(* IEC 61131-3 sources: plc-home-automation/home_automation/lighting_heating_updated, 19 files *)

(* ---- AlarmGlobals.st ---- *)
VAR_GLOBAL CONSTANT

   C_FRONT_DOOR_OPENING : INT := 1;
   C_GARAGE_DOOR_OPENING : UINT   := 2;
   C_HALL_ZONE : UINT        := 4;
   C_GARAGE_ZONE : UINT          := 5;
   C_KITCHEN_ZONE : UINT          := 6;
   C_LIVING_ROOM_ZONE : UINT         := 7;
   C_BEDROOM_ZONE : UINT            := 8;
   C_DOWNSTAIRS_BATH_ZONE : UINT      := 9;
   C_HALLWAY_ZONE : UINT         := 10;
   C_CHILDRENS_ROOM_3_ZONE : UINT   := 11;
   C_CHILDRENS_ROOM_1_ZONE : UINT   := 12;
   C_CHILDRENS_ROOM_2_ZONE : UINT   := 13;
   C_UPSTAIRS_BATH_ZONE : UINT     := 14;
   C_WC_ZONE : UINT              := 15;
   C_BOILER_ZONE : UINT           := 16;

   C_UNCONNECTED_NO_OP : UINT    := 3;

   C_ALARM_ZONES : UINT      := 16;
END_VAR

VAR_GLOBAL
    PARADOX_COM : fbPAR_DIG_EVOsystem;
    PARADOX_DATA : T_PAR_DIG_EVO_SYSTEM_DATA;
    ALARM_ZONES_INACTIVITY : ARRAY [1 .. C_ALARM_ZONES] OF BOOL;
    ALARM_ZONES_SABOTAGE : ARRAY [1 .. C_ALARM_ZONES] OF BOOL;
    ALARM_ZONES_ERROR : ARRAY [1 .. C_ALARM_ZONES] OF BOOL;
    ALARM_ACTIVE : BOOL;

    AWAY_TIMER: TON;

    TIME_AWAY_SHORT : TIME := T#20m;
    TIME_AWAY_LONG : TIME := T#60m;
    GONE_FOR_5_MINUTES : BOOL := FALSE;
    GONE_FOR_SHORT_TIME : BOOL := FALSE;
    GONE_FOR_LONG_TIME : BOOL := FALSE;
END_VAR

FUNCTION awayFromHomeFor : bool
  VAR_INPUT
    awayFor : TIME;  (*Tell me if motion sensors are inactive for that time. Max is 20 days.*)
  END_VAR

  IF(AWAY_TIMER.ET < awayFor) THEN
    awayFromHomeFor := false;
  ELSE
    awayFromHomeFor := true;
  END_IF;

END_FUNCTION

(* ---- HeatingGlobals.st ---- *)
VAR_GLOBAL CONSTANT
   // Heating control locals
   C_BEDROOM_INDEX : INT          := 0;
   C_LIVING_ROOM_1_INDEX : INT     := 1;
   C_LIVING_ROOM_2_INDEX : INT     := 2;
   C_LIVING_ROOM_3_INDEX : INT     := 3;
   C_DOWNSTAIRS_BATH_INDEX : INT    := 4;
   C_HALL_INDEX : INT      := 5;
   C_GARAGE_INDEX : INT        := 6;
   C_CHILDRENS_ROOM_1_INDEX : INT := 7;
   C_CHILDRENS_ROOM_2_INDEX : INT := 8;
   C_CHILDRENS_ROOM_3_INDEX : INT := 9;
   C_HALLWAY_INDEX : INT       := 10;
   C_BOILER_INDEX : INT         := 11;
   C_WC_INDEX : INT            := 12;
   C_UPSTAIRS_BATH_INDEX : INT   := 13;

   C_HEATING_ZONES : INT                  := 14;
   C_DOWNSTAIRS_ZONE_MAX_INDEX_PLUS_ONE : INT := 7;

   C_MAXIMUM_HEATING_TEMPERATURE : REAL := 38.0;
   C_MINIMUM_HEATING_TEMPERATURE : REAL := 28.0;

   C_MAXIMUM_HOT_WATER_TEMPERATURE : REAL := 62.0;
   C_MINIMUM_HOT_WATER_TEMPERATURE : REAL := 35.0;

END_VAR

VAR_GLOBAL
    heatingRequests : ARRAY [0 .. C_HEATING_ZONES - 1] OF BOOL;
END_VAR

VAR_GLOBAL
   HEATING_CONTROL_SAMPLING_TIME : TIME := T#10m;
   IPID_K : REAL := 0.0005;
   IPID_TI : REAL := 0.0001;
   IPID_TD : REAL := 12000;
   OVERSHOOT_HISTERESIS : REAL := 0.2;

   HEATING_ENABLE : BOOL := true;
   HOT_WATER_ENABLE : BOOL := true;
   PRESENCE_BASED_HEATING_CONTROL : BOOL := true;
   PRESENCE_BASED_HOT_WATER_ENABLE : BOOL := true;

   FUTOVIZ_TEMPERATURE : REAL              := 30.0;
   HOT_WATER_TEMPERATURE : REAL  := 42.0;

   LIVING_ROOM_DESIRED_TEMPERATURE : REAL       := 22.0;
   BEDROOM_DESIRED_TEMPERATURE : REAL     := 20.5;
   CHILDRENS_ROOM_1_DESIRED_TEMPERATURE : REAL := 22.0;
   CHILDRENS_ROOM_2_DESIRED_TEMPERATURE : REAL := 21.0;
   CHILDRENS_ROOM_3_DESIRED_TEMPERATURE : REAL := 21.0;
   DOWNSTAIRS_BATH_DESIRED_TEMPERATURE : REAL    := 21.0;
   UPSTAIRS_BATH_DESIRED_TEMPERATURE : REAL   := 21.0;
   GARAGE_DESIRED_TEMPERATURE : REAL        := 5.0;
   BOILER_DESIRED_TEMPERATURE : REAL         := 5.0;
   WC_DESIRED_TEMPERATURE : REAL            := 5.0;
   HALLWAY_DESIRED_TEMPERATURE : REAL       := 5.0;
   HALL_DESIRED_TEMPERATURE : REAL      := 21;

   // For testing purposes only
   WC_TEMPERATURE : REAL              := 30.0;
   HALLWAY_TEMPERATURE : REAL         := 30.0;
   BOILER_ROOM_TEMPERATURE : REAL           := 30.0;

   SUM_HEATING_REQUIREMENT : BOOL := false;
   SUM_HEATING_WATER_TEMPERATURE_REQUIREMENT : REAL := 0;

   MEASURED_TEMPERATURES : ARRAY [0 .. C_HEATING_ZONES - 1] OF PTR_TO REAL;
   DESIRED_TEMPERATURES : ARRAY [0 .. C_HEATING_ZONES - 1] OF PTR_TO REAL;
   VALVE_ACTUATORS : ARRAY [0 .. C_HEATING_ZONES - 1] OF PTR_TO BOOL;

   // You can't take the ADR() of a real const global...
   C_50_FOK : REAL := 50.0;
   C_4_FOK : REAL := 4.0;
END_VAR

(* ---- PersistGlobals.st ---- *)
VAR_GLOBAL CONSTANT
    C_REALS_TO_PERSIST : INT      := 18;
    C_BOOLS_TO_PERSIST : INT      := 4;
    C_PERSIST_DIRECTORY_ROOT : STRING := 'PERSIST';
    C_PERSIST_HEATING_IPID_SUBDIR : STRING := '';
    C_PERSIST_HEATING_SUBDIR : STRING := '/HEATING';
    C_PERSIST_ROOM_TEMPERATURE_SUBDIR : STRING := '/ROOMTMP';
    C_PERSIST_BOILER_CONTROL_SUBDIR : STRING := '/BOILERCT';
END_VAR

VAR_GLOBAL
    REALS_TO_PERSIST : ARRAY [1 .. C_REALS_TO_PERSIST] OF PTR_TO REAL;
    REALS_TO_PERSIST_DIRS : ARRAY [1 .. C_REALS_TO_PERSIST] OF STRING;
    REALS_TO_PERSIST_NAMES : ARRAY [1 .. C_REALS_TO_PERSIST] OF STRING;
    BOOLS_TO_PERSIST : ARRAY [1 .. C_BOOLS_TO_PERSIST] OF PTR_TO BOOL;
    BOOLS_TO_PERSIST_DIRS : ARRAY [1 .. C_BOOLS_TO_PERSIST] OF STRING;
    BOOLS_TO_PERSIST_NAMES : ARRAY [1 .. C_BOOLS_TO_PERSIST] OF STRING;
END_VAR

(* ---- VaillantGlobals.st ---- *)
VAR_GLOBAL
  VAILLANT_ACN                   : bool;  (*altered after loading all the data*)
  VAILLANT_HEATING_TEMP          : real;  (*current boiler temperature*)
  VAILLANT_DWH_TEMP              : real;  (*current DHW temperature*)
  VAILLANT_OUTSIDE_TEMP          : real;  (*current outdoor temperature on boiler sensor*)
  VAILLANT_RETURN_WATER_TEMP     : real;  (*current returning temperature (Some boilers don't measure it)*)
  VAILLANT_MODULATION_LEVEL      : usint; (*value of relative burner modulation (0-100%)*)
  VAILLANT_PRESSURE_LEVEL        : real;  (*value of pressure temperature water (0-5 bar)*)
  VAILLANT_BURNERS_RUNNING       : uint;  (*number of burner starts*)
  VAILLANT_HEATING_ACTIVE        : bool;  (*heating is active (heats right now)*)
  VAILLANT_DWH_ACTIVE            : bool;  (*DHW active (heats right now)*)
  VAILANT_DWH_PRESENT            : bool;  (*boiler reports DHW is present*)
  VAILANT_MODULATION_SUPPORT     : bool;  (*boiler supports power modulation*)
  VAILANT_BURNER_ON              : bool;  (*flame on*)
  VAILANT_ERROR                  : bool;  (*boiler has an error*)
  VAILLANT_DIAG_CODE             : uint;  (*diagnostic code boiler (lower byte = error code = upper byte error flags)*)
  VAILANT_COMMUNICATIONO_ERROR   : bool;  (*communication error*)

END_VAR

(* ---- BathroomFanOnOff.st ---- *)
FUNCTION logBathroomFan : INT
VAR_INPUT
    name : STRING;
    rampOn : BOOL;
    feedOn: BOOL;
    out : BOOL;
END_VAR
     SWITCH_TRACKER(name := name
         + ': ramp(' + BOOL_TO_STRING(rampOn)
         + ') feedOn(' + BOOL_TO_STRING(feedOn)
         + ') out(' + BOOL_TO_STRING(out)
         + ')');

    logBathroomFan := 0;
END_FUNCTION

FUNCTION_BLOCK BathroomFanOnOff

  VAR_INPUT CONSTANT
     name : STRING;
  END_VAR

  VAR_INPUT
     timeOn   : TIME;
     feedOn   : BOOL R_EDGE;
     feedOff  : BOOL R_EDGE;
     change   : BOOL R_EDGE;
  END_VAR

  VAR_OUTPUT
     out : BOOL;
  END_VAR

  VAR
     ramp    : TON;
     rampOn  : BOOL := false;
  END_VAR

  IF change THEN
     rampOn := NOT out;
     out := NOT out;
     logBathroomFan(name:= name, feedOn := feedOn, rampOn := rampOn, out := out);
  END_IF;

  IF feedOn THEN
     rampOn := false;
     out := true;
  END_IF;

  IF feedOff AND out THEN
     rampOn := true;
  END_IF;

  ramp(IN := rampOn, PT := timeOn);

  IF ramp.Q THEN
     out := false;
     rampOn := false;
  END_IF;

END_FUNCTION_BLOCK

(* ---- lighting.ST ---- *)
// Helper function block
TYPE
  ControllerArray : ARRAY [0 .. C_LIGHTS_ZONES_COUNT - 1] OF ChangeOnOff;
END_TYPE

FUNCTION_BLOCK TurnOffLightsHelper
  VAR_INPUT
    offSignal : BOOL R_EDGE;
  END_VAR

  VAR_IN_OUT
    controllers : ControllerArray;
  END_VAR

  VAR
    i : INT := 0;
  END_VAR

  IF (offSignal) THEN
    FOR i := 0 TO C_LIGHTS_ZONES_COUNT - 1 DO
      controllers[i](requestOff := offSignal);
    END_FOR;
  END_IF;

END_FUNCTION_BLOCK // Helper function block

PROGRAM LightingControl

  VAR
    domesticHotWaterCirculation_in : OnThenOffPulse;
    garageGate_in : OnThenOffPulse;

    exhaustRequest: BOOL := false;
    wcExhaustDelay : TON;
    wcExhaustDelayTime : TIME := T#4m;
    upstairsBathroomExhaustDelay : TON;
    upstairsBathroomExhaustDelayTime : TIME := T#8m;
    upstairsShowerExhaustDelay : TON;
    upstairsShowerExhaustDelayTime : TIME := T#3m;
    exhaustFan_in : BathroomFanOnOff;
    exhaustFanRuntime : TIME := T#10m;

    lightsKapcsolok : ControllerArray;
    lightsControlBasedOnOccupancy : TurnOffLightsHelper;

    i : INT := 0;

  END_VAR

    KITCHEN_FURNITURE_LIGHTS_OUT := TRUE; // We have the door bell in that socket for now.

    domesticHotWaterCirculation_in(timeOn := T#2m, timeOff := T#20m, onSignal := (KERINTGETES_SWITCH_IN OR KITCHEN_FURNITURE_LIGHTS_IN OR VIRTUAL_CIRCULATION_SWITCH_IN));
    BOILER_PUMP_PLUG_RIGHT := domesticHotWaterCirculation_in.active;
    VIRTUAL_CIRCULATION_SWITCH_IN := FALSE;

    wcExhaustDelay(IN := UPSTAIRS_WC_LIGHTS_OUT, PT := wcExhaustDelayTime);
    upstairsBathroomExhaustDelay(IN := UPSTAIRS_BATH_MAJOR_LIGHTS_OUT, PT := upstairsBathroomExhaustDelayTime);
    upstairsShowerExhaustDelay(IN := UPSTAIRS_BATH_SHOWER_LIGHTS_OUT, PT := upstairsShowerExhaustDelayTime);
    //exhaustRequest := wcExhaustDelay.Q OR upstairsBathroomExhaustDelay.Q OR upstairsShowerExhaustDelay.Q;
    exhaustRequest := FALSE;
    exhaustFan_in(timeOn := exhaustFanRuntime, feedOn := exhaustRequest, feedOff := NOT exhaustRequest, change := EXHAUST_FAN_IN OR VIRTUAL_EXHAUST_FAN_IN, name := 'Elszivo ventillator');
    EXHAUST_FAN_OUT := exhaustFan_in.out;
    VIRTUAL_EXHAUST_FAN_IN := FALSE;

    garageGate_in(onSignal := GARAGE_GATE_IN OR VIRTUAL_GARAGE_DOOR_OPENER, timeOn := T#0.2s, timeOff := T#0.2s);
    GARAGE_GATE_OUT := garageGate_in.active;
    VIRTUAL_GARAGE_DOOR_OPENER := FALSE;

    HALLWAY_LIGHTS_COMBINED_IN := HALLWAY_LIGHTS_IN OR STAIRS_LIGHTS_IN;

    FOR i := 0 TO C_LIGHTS_ZONES_COUNT - 1 DO
        lightsKapcsolok[i](requestChange := ( LIGHTS_INPUTS[i]^ OR VIRTUAL_LIGHTS_INPUTS[i]^) );
        LIGHTS_OUTPUTS[i]^ := lightsKapcsolok[i].output;
        VIRTUAL_LIGHTS_INPUTS[i]^ := FALSE;
    END_FOR;

    lightsControlBasedOnOccupancy( offSignal := (ALARM_ACTIVE AND GONE_FOR_SHORT_TIME), controllers := lightsKapcsolok );

END_PROGRAM

(* ---- LinearHeatController.st ---- *)
FUNCTION_BLOCK LinearHeatController
  VAR_INPUT
    actualTemperature : REAL := 0;
    setpoint : REAL := 0;
    ramp : REAL := 1;
    offset : REAL := 0;
    histeresis : REAL := 0;
  END_VAR
  VAR_OUTPUT
    heatRequest : BOOL := FALSE;
    heatingTemperature : REAL := 0;
  END_VAR

  heatingTemperature := setpoint + ramp * (setpoint - actualTemperature) + offset;

  IF actualTemperature < (setpoint - histeresis) THEN
     heatRequest := true;
  END_IF;
  IF actualTemperature > (setpoint + histeresis) THEN
     heatRequest := FALSE;
  END_IF;
END_FUNCTION_BLOCK

(* ---- PersistFramework.st ---- *)
FUNCTION createDirectory: BOOL
VAR_INPUT
    dirPath: STRING;
END_VAR

VAR
    errorMessage: STRING;

END_VAR

createDirectory := FileExists(fileName := dirPath);
IF NOT createDirectory THEN
  createDirectory := DirCreate(dirName := dirPath);
  IF NOT createDirectory THEN
    GetLastErrTxt( errCode := GetLastErr(), errMessage := errorMessage);
    FILE_PROBLEM_TRACKER(name := 'Dir create error:');
    FILE_PROBLEM_TRACKER(name := dirPath);
    FILE_PROBLEM_TRACKER(name := errorMessage);
    return;
  END_IF;
END_IF;

createDirectory := true;

END_FUNCTION

FUNCTION_BLOCK Persistor

VAR_IN_OUT
    compilerBugPlaceholder: BOOL;
    dirPath: STRING;
    fileName: STRING;
    data : UDINT;
END_VAR
VAR_INPUT
    dataSize: UDINT;
    toWrite : BOOL;
END_VAR
VAR_OUTPUT
    busy: BOOL := FALSE;
END_VAR

VAR
    fullPath : STRING;

    writer  : WriteToFile;
    reader : ReadFromFile;
    reading : BOOL := false;
    writing : BOOL := false;

    errorMessage : STRING;
    file : BOOL;
END_VAR

// Workaround for a compiler bug which renders the address of the first VAR_IN_OUT to the unusable %X0.0 no matter what.
IF FALSE THEN compilerBugPlaceholder := compilerBugPlaceholder; END_IF;

IF writing THEN
    writer( fileName := fullPath,
            srcVar := data,
            exec := writing,
            seek := 0,
            size := dataSize
            );
    writing := writer.busy;
    IF writer.err THEN
      GetLastErrTxt(errCode := writer.errID, errMessage := errorMessage);
      FILE_PROBLEM_TRACKER(name := 'File write error: ');
      FILE_PROBLEM_TRACKER(name := fullPath);
      FILE_PROBLEM_TRACKER(name := errorMessage);
      return;
    END_IF;

ELSIF reading THEN
    reader( fileName := fullPath,
            dstVar := data,
            exec := reading,
            seek := 0,
            size := dataSize
            );
    reading := reader.busy;
    IF reader.err THEN
      GetLastErrTxt(errCode := writer.errID, errMessage := errorMessage);
      FILE_PROBLEM_TRACKER(name := 'Read error:');
      FILE_PROBLEM_TRACKER(name := fullPath);
      FILE_PROBLEM_TRACKER(name := errorMessage);
      return;
    END_IF;

ELSE

    fullPath := dirPath + '/' + fileName;

    IF toWrite THEN
      createDirectory(dirPath := dirPath);

      IO_LOGGER(name := 'Writing to file: ');
      IO_LOGGER(name := dirPath);
      IO_LOGGER(name := fileName);

      writer( fileName := fullPath, srcVar := data, exec := writing, seek := 0, size := dataSize ); // For the sake of edge
      writing := TRUE;

    ELSE  // toRead
      file := FileExists(fileName := fullPath);
      IF NOT file THEN
        GetLastErrTxt(errCode := GetLastErr(), errMessage := errorMessage);
        FILE_PROBLEM_TRACKER(name := 'Can not find file to read: ');
        FILE_PROBLEM_TRACKER(name := fullPath);
        FILE_PROBLEM_TRACKER(name := errorMessage);
        return;
      END_IF;

      IO_LOGGER(name := 'Reading from file: ');
      IO_LOGGER(name := dirPath);
      IO_LOGGER(name := fileName);

      reader( fileName := fullPath, dstVar := data, exec := writing, seek := 0, size := dataSize ); // For the sake of edge
      reading := TRUE;
    END_IF;
END_IF;

busy := reading OR writing;

END_FUNCTION_BLOCK // Persistor

// -------------------------------------------------------------------------------------

FUNCTION_BLOCK PersistBool

VAR_IN_OUT
    compilerBugPlaceholder: BOOL;
    variableToPersist : BOOL;
    dirPath : STRING;
    fileName : STRING;
END_VAR
VAR_INPUT
    toWrite : BOOL;
END_VAR
VAR_OUTPUT
END_VAR
VAR
    persistImpl: Persistor;
    current: BOOL;
    previous: BOOL;
    actionIsWrite : BOOL;

    variableAsString : STRING[1];
END_VAR

// Workaround for a compiler bug which renders the address of the first VAR_IN_OUT to the unusable %X0.0 no matter what.
IF FALSE THEN compilerBugPlaceholder := compilerBugPlaceholder; END_IF;

IF NOT persistImpl.busy THEN
  previous := current;
  current := variableToPersist;
  actionIsWrite := toWrite;
END_IF;

IF actionIsWrite THEN
  IF NOT (current = previous) THEN
    variableAsString := BOOL_TO_STRING(current);
    persistImpl(compilerBugPlaceholder := compilerBugPlaceholder,
       dirPath := dirPath,
       fileName := fileName,
       data := void(variableAsString),
       dataSize := SIZEOF(variableAsString),
       toWrite := toWrite);
    IF NOT persistImpl.busy THEN
      IO_LOGGER(name := 'Wrote value:');
      IO_LOGGER(name := variableAsString);
    END_IF;
  END_IF;
ELSE

  persistImpl(compilerBugPlaceholder := compilerBugPlaceholder,
     dirPath := dirPath,
     fileName := fileName,
     data := void(variableAsString),
     dataSize := SIZEOF(variableAsString),
     toWrite := toWrite);
  IF NOT persistImpl.busy THEN
    IO_LOGGER(name := 'Read value');
    IO_LOGGER(name := variableAsString);
    variableToPersist := STRING_TO_BOOL(variableAsString);
    current := variableToPersist;
  END_IF;
END_IF;

END_FUNCTION_BLOCK // PersistBool

// -------------------------------------------------------------------------------------

FUNCTION_BLOCK PersistReal

VAR_IN_OUT
    compilerBugPlaceholder: BOOL;
    variableToPersist : REAL;
    dirPath : STRING;
    fileName : STRING;
END_VAR
VAR_INPUT
    toWrite : BOOL;
END_VAR
VAR_OUTPUT
END_VAR
VAR
    persistImpl: Persistor;
    current: REAL;
    previous: REAL;
    actionIsWrite : BOOL;

    variableAsString : STRING;
END_VAR

// Workaround for a compiler bug which renders the address of the first VAR_IN_OUT to the unusable %X0.0 no matter what.
IF FALSE THEN compilerBugPlaceholder := compilerBugPlaceholder; END_IF;

IF NOT persistImpl.busy THEN
  previous := current;
  current := variableToPersist;
  actionIsWrite := toWrite;
END_IF;

IF actionIsWrite THEN
  IF NOT (current = previous) THEN
    variableAsString := REAL_TO_STRING(current);
    persistImpl(compilerBugPlaceholder := compilerBugPlaceholder,
       dirPath := dirPath,
       fileName := fileName,
       data := void(current),
       dataSize := SIZEOF(current),
       toWrite := toWrite);
    IF NOT persistImpl.busy THEN
      IO_LOGGER(name := 'Wrote value as binary:');
      IO_LOGGER(name := variableAsString);
    END_IF;
  END_IF;
ELSE

  persistImpl(compilerBugPlaceholder := compilerBugPlaceholder,
     dirPath := dirPath,
     fileName := fileName,
     data := void(current),
     dataSize := SIZEOF(current),
     toWrite := toWrite);
  IF NOT persistImpl.busy THEN
    variableAsString := REAL_TO_STRING(current);
    IO_LOGGER(name := 'Read value from binary:');
    IO_LOGGER(name := variableAsString);
    variableToPersist := current;
  END_IF;
END_IF;

END_FUNCTION_BLOCK // PersistReal

(* ---- PidController.st ---- *)
FUNCTION_BLOCK IPidController

    VAR_INPUT
        setpoint: REAL;
        actual: REAL;
        previousControlledProperty : REAL;
        samplingTime: TIME;

        k : REAL;
        tI: REAL; // In seconds
        tD: REAL; // In seconds

        previousIntegrationError : REAL;
    END_VAR

    VAR_OUTPUT
        integrationError : REAL;
        controlledProperty : REAL;
    END_VAR

    VAR
        samplingTimer : TON;
        error: REAL := 0;
        timePassed : REAL; // In seconds
        lastError : REAL;
    END_VAR

    samplingTimer(IN := true, PT := samplingTime);
    IF samplingTimer.Q THEN
        timePassed := TIME_TO_REAL(samplingTime) / 1000;

        samplingTimer(IN := false, PT := samplingTime);
        samplingTimer(IN := true, PT := samplingTime);

        error := setpoint - actual;
        integrationError := (previousIntegrationError + error) * tI * timePassed;

        controlledProperty := previousControlledProperty
                              + k * error * timePassed
                              + integrationError
                              + (error - lastError) / timePassed * tD;

        lastError := error;
    END_IF;

END_FUNCTION_BLOCK

(* ---- PidHeatController.st ---- *)
FUNCTION_BLOCK IPidHeatController

VAR_INPUT
    actualTemperature: REAL;
    setpoint: REAL;
    samplingTime: TIME;
    actualHeatingTemperature: REAL;

    minimumHeatingTemperature : REAL;
    maximumHeatingTemparature : REAL;

    k : REAL;
    tI: REAL; // In seconds
    tD: REAL; // In seconds

    overshootHisteresis : REAL;
END_VAR

VAR_OUTPUT
    heatRequest : BOOL := false;
    heatingTemperature : REAL := 0;
END_VAR

VAR
    integrationError : REAL := 0;
    ipid : IPidController;
END_VAR

    IF actualTemperature > (setpoint + overshootHisteresis) THEN
        heatRequest := false;
    ELSIF actualTemperature < (setpoint - overshootHisteresis) THEN
        heatRequest := true;
    END_IF;

    IF heatRequest THEN
        ipid(setpoint := setpoint,
            actual := actualTemperature,
            previousControlledProperty := actualHeatingTemperature,
            samplingTime := samplingTime,
            k := k,
            tI := tI,
            tD := tD,
            previousIntegrationError := integrationError);
        integrationError := ipid.integrationError;
    END_IF;

    IF ipid.controlledProperty > maximumHeatingTemparature THEN
        heatingTemperature := maximumHeatingTemparature;
    ELSIF ipid.controlledProperty < minimumHeatingTemperature THEN
        heatingTemperature := minimumHeatingTemperature;
    ELSE
        heatingTemperature := ipid.controlledProperty;
    END_IF;

END_FUNCTION_BLOCK

(* ---- StringRecorder.st ---- *)
VAR_GLOBAL CONSTANT
  C_BUFFER_SIZE : INT := 20;
  C_STRING_SIZE : INT := 200;
END_VAR

FUNCTION_BLOCK StringRecorder
  VAR
    whoTouchedMe : ARRAY [1..C_BUFFER_SIZE] OF STRING[C_STRING_SIZE];
    touchIndex: INT := 0;
  END_VAR
  VAR_INPUT
    name: STRING;
  END_VAR

  IF touchIndex = C_BUFFER_SIZE THEN
      touchIndex := 1;
  ELSE
      touchIndex := touchIndex + 1;
  END_IF;
  whoTouchedMe[touchIndex] := LEFT(IN := name, L := C_STRING_SIZE - 1);

END_FUNCTION_BLOCK

VAR_GLOBAL
  SWITCH_TRACKER : StringRecorder;
  FILE_PROBLEM_TRACKER : StringRecorder;
  IO_LOGGER : StringRecorder;
END_VAR

(* ---- TimeSwitch.st ---- *)
FUNCTION_BLOCK TimeSwitchImpl
  VAR_INPUT CONSTANT
    name : STRING;
  END_VAR

  VAR_INPUT
    onSignal : BOOL R_EDGE;
    offSignal : BOOL R_EDGE;
    maxDuration: TIME := T#1m;
  END_VAR

  VAR_OUTPUT
    active : BOOL := FALSE;
    duration : TIME := T#0s;
  END_VAR

  VAR
    timer : TON;
  END_VAR

  IF onSignal THEN
     active := TRUE;
  END_IF;

  IF active THEN
     timer(IN := TRUE, PT := maxDuration);
  END_IF;

  IF offSignal THEN
     active := FALSE;
     duration := timer.ET;
     timer(IN := FALSE);
     SWITCH_TRACKER(name := name + TIME_TO_STRING(duration));
  END_IF;
END_FUNCTION_BLOCK

FUNCTION_BLOCK TimeSwitch

  VAR_INPUT CONSTANT
    name : STRING;
  END_VAR

  VAR_INPUT
    onSignal : bool;
    maxDuration: TIME;
  END_VAR

  VAR_OUTPUT
    active : BOOL := FALSE;
    duration : TIME := T#0s;
  END_VAR

  VAR
    impl : TimeSwitchImpl;
  END_VAR

  impl(onSignal := onSignal, offSignal := NOT onSignal, maxDuration := maxDuration, name := name);
  active := impl.active;
  duration := impl.duration;

END_FUNCTION_BLOCK

(* ---- Alarm.ST ---- *)
PROGRAM AlarmControl
  VAR_INPUT
  END_VAR
  VAR_OUTPUT
  END_VAR
  VAR
     i: UINT;
     sumAktivitas : BOOL := FALSE;
     heatingVezerles : InPlaceOnOff;
     melegVizVezerles : InPlaceOnOff;

     heatingVezerloNev : STRING := 'Alarm heating control';
     melegVizVezerloNev : STRING := 'Alarm meleg viz control';
  END_VAR

  alarmRead();

  // Turn on warm water circulation when someone enters through the entrance doors after the alarm cooldown time.
  VIRTUAL_CIRCULATION_SWITCH_IN := GONE_FOR_SHORT_TIME AND
      (NOT ALARM_ZONES_INACTIVITY[C_GARAGE_DOOR_OPENING] OR NOT ALARM_ZONES_INACTIVITY[C_FRONT_DOOR_OPENING]);

  // Detecting if house is no longer occupied or everyone is sleeping
  sumAktivitas := FALSE;
  FOR i := 1 TO C_ALARM_ZONES DO
      sumAktivitas := sumAktivitas OR (NOT ALARM_ZONES_INACTIVITY[i]);
  END_FOR;
  AWAY_TIMER(IN := NOT sumAktivitas, PT := T#20d);
  GONE_FOR_5_MINUTES := awayFromHomeFor(awayFor := T#5m);
  GONE_FOR_SHORT_TIME := awayFromHomeFor(TIME_AWAY_SHORT);
  GONE_FOR_LONG_TIME := awayFromHomeFor(TIME_AWAY_LONG);

  IF PRESENCE_BASED_HEATING_CONTROL THEN
     heatingVezerles(onSignal := NOT GONE_FOR_LONG_TIME,
         offSignal := ((ALARM_ACTIVE AND GONE_FOR_5_MINUTES) OR GONE_FOR_LONG_TIME),
         name := heatingVezerloNev,
         controlledVariable := HEATING_ENABLE);
  END_IF;
  IF PRESENCE_BASED_HOT_WATER_ENABLE THEN
     melegVizVezerles(onSignal := NOT GONE_FOR_SHORT_TIME,
         offSignal := ((ALARM_ACTIVE AND GONE_FOR_5_MINUTES) OR GONE_FOR_SHORT_TIME),
         name := melegVizVezerloNev,
         controlledVariable := HOT_WATER_ENABLE);
  END_IF;

END_PROGRAM

(* ---- heating.ST ---- *)
PROGRAM HeatingControl
(*Controlling Vaillant Exotec Exclusive heating bioler over VR33 OpenTherm card using tecomat OpenTherm unit.
*)

  VAR
    // Techincals for OpenThem communication
    vaillant_opentherm : fbOpenTherm;
    commEnable : BOOL := true;

    termosztatok : ARRAY [0 .. C_HEATING_ZONES - 1] OF IPidHeatController;
    eloremenoVizhoRequests : ARRAY [0 .. C_HEATING_ZONES - 1] OF REAL;

    // Boiler heating state
    heating_inditas : BOOL := false;

    i : INT := 0;
    activeZones : REAL := 0;

    downstairsPumpRequest : BOOL := false;
    upstairsPumpRequest : BOOL := false;
    downstairsPumpActivationIdozito: TON;
    upstairsPumpActivationIdozito: TON;
    downstairsPumpDeactivationIdozito : TOF;
    upstairsPumpDeactivationIdozito : TOF;
    pumpActivationDelay : TIME := T#10m;
    pumpDeactivationDelay : TIME := T#1m;

  END_VAR

    // Eredõ vezérlés
    SUM_HEATING_REQUIREMENT := false;
    downstairsPumpRequest := false;
    upstairsPumpRequest := false;
    SUM_HEATING_WATER_TEMPERATURE_REQUIREMENT := 0;
    activeZones := 0;

    // Keep heating water temperature within limits
    IF HOT_WATER_TEMPERATURE > C_MAXIMUM_HOT_WATER_TEMPERATURE THEN
       HOT_WATER_TEMPERATURE := C_MAXIMUM_HOT_WATER_TEMPERATURE;
    END_IF;

    IF HOT_WATER_TEMPERATURE < C_MINIMUM_HOT_WATER_TEMPERATURE THEN
       HOT_WATER_TEMPERATURE := C_MINIMUM_HOT_WATER_TEMPERATURE;
    END_IF;

    FOR i := 0 TO C_HEATING_ZONES - 1 DO
        // avoid unlimited accumlation of integrative error
        IF HEATING_ENABLE THEN
            termosztatok[i](
                actualTemperature := MEASURED_TEMPERATURES[i]^,
                setpoint := DESIRED_TEMPERATURES[i]^,
                actualHeatingTemperature := eloremenoVizhoRequests[i],
                samplingTime := HEATING_CONTROL_SAMPLING_TIME,
                k := IPID_K,
                tI := IPID_TI,
                tD := IPID_TD,
                minimumHeatingTemperature := C_MINIMUM_HEATING_TEMPERATURE,
                maximumHeatingTemparature := C_MAXIMUM_HEATING_TEMPERATURE,
                overshootHisteresis := OVERSHOOT_HISTERESIS
            );
        END_IF;
        // Enable heat request for a zone only if global control flag is enabled
        heatingRequests[i] := termosztatok[i].heatRequest AND HEATING_ENABLE;
        eloremenoVizhoRequests[i] := termosztatok[i].heatingTemperature;
        SUM_HEATING_REQUIREMENT := SUM_HEATING_REQUIREMENT OR heatingRequests[i];
        IF heatingRequests[i] THEN
            SUM_HEATING_WATER_TEMPERATURE_REQUIREMENT := SUM_HEATING_WATER_TEMPERATURE_REQUIREMENT + eloremenoVizhoRequests[i];
            activeZones := activeZones + 1;
        END_IF;

        IF heatingRequests[i] THEN
            IF i < C_DOWNSTAIRS_ZONE_MAX_INDEX_PLUS_ONE THEN
                downstairsPumpRequest := true;
            ELSE
                upstairsPumpRequest := true;
            END_IF;
        END_IF;
    END_FOR;

    IF activeZones > 0 THEN
       SUM_HEATING_WATER_TEMPERATURE_REQUIREMENT := SUM_HEATING_WATER_TEMPERATURE_REQUIREMENT / activeZones;
    END_IF;

    // Control valves
    FOR i := 0 TO C_HEATING_ZONES - 1 DO
        IF i < C_DOWNSTAIRS_ZONE_MAX_INDEX_PLUS_ONE THEN
            IF i = C_GARAGE_INDEX THEN
                // Tis is a normally closed valve
                VALVE_ACTUATORS[i]^ := heatingRequests[i] AND downstairsPumpRequest;
            ELSE
                VALVE_ACTUATORS[i]^ := NOT heatingRequests[i] AND downstairsPumpRequest;
            END_IF;
        ELSE
            VALVE_ACTUATORS[i]^ := NOT heatingRequests[i] AND upstairsPumpRequest;
        END_IF;
    END_FOR;

    downstairsPumpActivationIdozito(IN := downstairsPumpRequest, PT := pumpActivationDelay);
    downstairsPumpDeactivationIdozito(IN := downstairsPumpActivationIdozito.Q, PT := pumpDeactivationDelay);
    upstairsPumpActivationIdozito(IN := upstairsPumpRequest, PT := pumpActivationDelay);
    upstairsPumpDeactivationIdozito(IN := upstairsPumpActivationIdozito.Q, PT := pumpActivationDelay);

    STORAGE_PUMP := downstairsPumpDeactivationIdozito.Q;
    BOILER_PUMP_PLUG_LEFT := upstairsPumpDeactivationIdozito.Q;

    futoviz_temperature := SUM_HEATING_WATER_TEMPERATURE_REQUIREMENT;
    heating_inditas := downstairsPumpActivationIdozito.Q OR upstairsPumpActivationIdozito.Q;

    // Actual OpenTherm communication
    vaillant_opentherm(
      in_communicate := commEnable,
      in_CH_en := heating_inditas AND HEATING_ENABLE,
      in_DHW_en := HOT_WATER_ENABLE,
      in_CH_temp := futoviz_temperature,
      in_max_CH_temp := C_MAXIMUM_HEATING_TEMPERATURE,
      in_DHW_temp := HOT_WATER_TEMPERATURE,
      in_timeOut := T#10s,
      in_timeIdle := T#5s,
      UC1204_IN := void(OPENTHERM_IN),
      UC1204_OUT := void(OPENTHERM_OUT),
      OT_COMM_ARRAY := void(OT_COMM_ARRAY_GEMINOX_THRI)
    ); // Vailant Ecotec Exclusive should support all OT oiperations

    VAILLANT_ACN := vaillant_opentherm.out_ACN;
    VAILLANT_HEATING_TEMP := vaillant_opentherm.out_heating_temp;
    VAILLANT_DWH_TEMP  := vaillant_opentherm.out_DHW_temp;
    VAILLANT_OUTSIDE_TEMP := vaillant_opentherm.out_outside_temp;
    VAILLANT_RETURN_WATER_TEMP := vaillant_opentherm.out_ret_water_temp;
    VAILLANT_MODULATION_LEVEL := vaillant_opentherm.out_modulation_level;
    VAILLANT_PRESSURE_LEVEL := vaillant_opentherm.out_pressure_level;
    VAILLANT_BURNERS_RUNNING := vaillant_opentherm.out_burner_starts;
    VAILLANT_HEATING_ACTIVE := vaillant_opentherm.out_CH_active;
    VAILLANT_DWH_ACTIVE := vaillant_opentherm.out_DHW_active;
    VAILANT_DWH_PRESENT := vaillant_opentherm.out_DHW_present;
    VAILANT_MODULATION_SUPPORT := vaillant_opentherm.out_modulating;
    VAILANT_BURNER_ON := vaillant_opentherm.out_flame;
    VAILANT_ERROR := vaillant_opentherm.out_com_error;
    VAILLANT_DIAG_CODE := vaillant_opentherm.out_diag_code;
    VAILANT_COMMUNICATIONO_ERROR := vaillant_opentherm.out_com_error;

(*
  timer(IN := true, PT := T#5s);
  IF timer.Q THEN
    UcOut.cont.ACN := ack;
    UcOut.MSG_TYPE := 0;
    UcOut.DATA_ID := dataID;
    UcOut.DATA_VAL := 0;
    VAILLANT_OPENTHERM_OUT := UcOut;
    UcIn := VAILLANT_OPENTHERM_IN;
    timer(IN := false, PT := T#5s);
  END_IF;
 *)

END_PROGRAM

(* ---- HeatingInint.ST ---- *)
PROGRAM HeatingInint
  VAR
     initialised : BOOL := false;
  END_VAR

  IF initialised = false THEN
      initialised := true;

      MEASURED_TEMPERATURES[C_BEDROOM_INDEX] := ADR(BEDROOM_TEMPERATURE);
      MEASURED_TEMPERATURES[C_LIVING_ROOM_1_INDEX] := ADR(LIVING_ROOM_TEMPERATURE);
      MEASURED_TEMPERATURES[C_LIVING_ROOM_2_INDEX] := ADR(LIVING_ROOM_TEMPERATURE);
      MEASURED_TEMPERATURES[C_LIVING_ROOM_3_INDEX] := ADR(LIVING_ROOM_TEMPERATURE);
      MEASURED_TEMPERATURES[C_DOWNSTAIRS_BATH_INDEX] := ADR(DOWNSTAIRS_BATH_TEMPERATURE);
      MEASURED_TEMPERATURES[C_HALL_INDEX] := ADR(HALL_TEMPERATURE);
      MEASURED_TEMPERATURES[C_GARAGE_INDEX] := ADR(GARAGE_TEMPERATURE);
      MEASURED_TEMPERATURES[C_CHILDRENS_ROOM_1_INDEX] := ADR(CHILDRENS_ROOM_1_TEMPERATURE);
      MEASURED_TEMPERATURES[C_CHILDRENS_ROOM_2_INDEX] := ADR(CHILDRENS_ROOM_2_TEMPERATURE);
      MEASURED_TEMPERATURES[C_CHILDRENS_ROOM_3_INDEX] := ADR(CHILDRENS_ROOM_3_TEMPERATURE);
      MEASURED_TEMPERATURES[C_HALLWAY_INDEX] := ADR(HALLWAY_TEMPERATURE);
      MEASURED_TEMPERATURES[C_BOILER_INDEX] := ADR(BOILER_ROOM_TEMPERATURE);
      MEASURED_TEMPERATURES[C_WC_INDEX] := ADR(WC_TEMPERATURE);
      MEASURED_TEMPERATURES[C_UPSTAIRS_BATH_INDEX] := ADR(UPSTAIRS_BATH_TEMPERATURE);

      DESIRED_TEMPERATURES[C_BEDROOM_INDEX] := ADR(BEDROOM_DESIRED_TEMPERATURE);
      DESIRED_TEMPERATURES[C_LIVING_ROOM_1_INDEX] := ADR(LIVING_ROOM_DESIRED_TEMPERATURE);
      DESIRED_TEMPERATURES[C_LIVING_ROOM_2_INDEX] := ADR(LIVING_ROOM_DESIRED_TEMPERATURE);
      DESIRED_TEMPERATURES[C_LIVING_ROOM_3_INDEX] := ADR(LIVING_ROOM_DESIRED_TEMPERATURE);
      DESIRED_TEMPERATURES[C_DOWNSTAIRS_BATH_INDEX] := ADR(DOWNSTAIRS_BATH_DESIRED_TEMPERATURE);
      DESIRED_TEMPERATURES[C_HALL_INDEX] := ADR(HALL_DESIRED_TEMPERATURE);
      DESIRED_TEMPERATURES[C_GARAGE_INDEX] := ADR(GARAGE_DESIRED_TEMPERATURE);
      DESIRED_TEMPERATURES[C_CHILDRENS_ROOM_1_INDEX] := ADR(CHILDRENS_ROOM_1_DESIRED_TEMPERATURE);
      DESIRED_TEMPERATURES[C_CHILDRENS_ROOM_2_INDEX] := ADR(CHILDRENS_ROOM_2_DESIRED_TEMPERATURE);
      DESIRED_TEMPERATURES[C_CHILDRENS_ROOM_3_INDEX] := ADR(CHILDRENS_ROOM_3_DESIRED_TEMPERATURE);
      DESIRED_TEMPERATURES[C_HALLWAY_INDEX] := ADR(HALLWAY_DESIRED_TEMPERATURE);
      DESIRED_TEMPERATURES[C_BOILER_INDEX] := ADR(BOILER_DESIRED_TEMPERATURE);
      DESIRED_TEMPERATURES[C_WC_INDEX] := ADR(WC_DESIRED_TEMPERATURE);
      DESIRED_TEMPERATURES[C_UPSTAIRS_BATH_INDEX] := ADR(UPSTAIRS_BATH_DESIRED_TEMPERATURE);

      VALVE_ACTUATORS[C_BEDROOM_INDEX] := ADR(BEDROOM_TERMOFEJ);
      VALVE_ACTUATORS[C_LIVING_ROOM_1_INDEX] := ADR(LIVING_ROOM_1_TERMOFEJ);
      VALVE_ACTUATORS[C_LIVING_ROOM_2_INDEX] := ADR(LIVING_ROOM_2_TERMOFEJ);
      VALVE_ACTUATORS[C_LIVING_ROOM_3_INDEX] := ADR(LIVING_ROOM_3_TERMOFEJ);
      VALVE_ACTUATORS[C_DOWNSTAIRS_BATH_INDEX] := ADR(DOWNSTAIRS_BATH_TERMOFEJ);
      VALVE_ACTUATORS[C_HALL_INDEX] := ADR(ELOSZABA_TERMOFEJ);
      VALVE_ACTUATORS[C_GARAGE_INDEX] := ADR(GARAGE_TERMOFEJ);
      VALVE_ACTUATORS[C_CHILDRENS_ROOM_1_INDEX] := ADR(CHILDRENS_ROOM_1_TERMOFEJ);
      VALVE_ACTUATORS[C_CHILDRENS_ROOM_2_INDEX] := ADR(CHILDRENS_ROOM_2_TERMOFEJ);
      VALVE_ACTUATORS[C_CHILDRENS_ROOM_3_INDEX] := ADR(CHILDRENS_ROOM_3_TERMOFEJ);
      VALVE_ACTUATORS[C_HALLWAY_INDEX] := ADR(HALLWAY_TERMOFEJ);
      VALVE_ACTUATORS[C_BOILER_INDEX] := ADR(BOILER_TERMOFEJ);
      VALVE_ACTUATORS[C_WC_INDEX] := ADR(WC_TERMOFEJ);
      VALVE_ACTUATORS[C_UPSTAIRS_BATH_INDEX] := ADR(UPSTAIRS_BATH_TERMOFEJ);

  END_IF;

END_PROGRAM

(* ---- LightingInit.st ---- *)
PROGRAM LightingInit

    VAR
        initialised : BOOL := false;
    END_VAR;

    IF initialised = FALSE THEN
        initialised := TRUE;

        LIGHTS_INPUTS[C_DOWNSTAIRS_BATH_MAJOR_LIGHTS_INDEX]     := ADR(DOWNSTAIRS_BATH_MAJOR_LIGHTS_IN);
        LIGHTS_INPUTS[C_DOWNSTAIRS_BATH_SHOWER_LIGHTS_INDEX]   := ADR(DOWNSTAIRS_BATH_SHOWER_LIGHTS_IN);
        LIGHTS_INPUTS[C_UPSTAIRS_BATH_MAJOR_LIGHTS_INDEX]    := ADR(UPSTAIRS_BATH_MAJOR_LIGHTS_IN);
        LIGHTS_INPUTS[C_UPSTAIRS_WC_LIGHTS_INDEX]            := ADR(UPSTAIRS_WC_VIALGITAS_IN);
        LIGHTS_INPUTS[C_UPSTAIRS_BATH_SHOWER_LIGHTS_INDEX]  := ADR(UPSTAIRS_BATH_SHOWER_LIGHTS_IN);
        LIGHTS_INPUTS[C_OUTDOOR_LIGHTS_INDEX]             := ADR(OUTDOOR_LIGHTS_IN);
        LIGHTS_INPUTS[C_HALL_LIGHTS_INDEX]            := ADR(HALL_LIGHTS_IN);
        LIGHTS_INPUTS[C_GARAGE_LIGHTS_INDEX]              := ADR(GARAGE_LIGHTS_IN);
        LIGHTS_INPUTS[C_MAJOR_STORAGE_LIGHTS_INDEX]         := ADR(MAJOR_STORAGE_LIGHTS_IN);
        LIGHTS_INPUTS[C_MINOR_STORAGE_LIGHTS_INDEX]          := ADR(MINOR_STORAGE_LIGHTS_IN);
        LIGHTS_INPUTS[C_GARDEN_BALCONY_LIGHTS_INDEX]        := ADR(GARDEN_BALCONY_LIGHTS_IN);
        LIGHTS_INPUTS[C_CHILDRENS_ROOM_2_LIGHTS_INDEX]       := ADR(CHILDRENS_ROOM_2_LIGHTS_IN);
        LIGHTS_INPUTS[C_CHILDRENS_ROOM_1_OUTER_LIGHTS_INDEX] := ADR(CHILDRENS_ROOM_1_OUTER_LIGHTS_IN);
        LIGHTS_INPUTS[C_CHILDRENS_ROOM_1_INNER_LIGHTS_INDEX] := ADR(CHILDRENS_ROOM_1_INNER_LIGHTS_IN);
        LIGHTS_INPUTS[C_CHILDRENS_ROOM_3_LIGHTS_INDEX]       := ADR(CHILDRENS_ROOM_3_LIGHTS_IN);
        LIGHTS_INPUTS[C_GATE_BALCONY_LIGHTS_INDEX]         := ADR(GATE_BALCONY_LIGHTS_IN);
        LIGHTS_INPUTS[C_DOWNSTAIRS_BEDROOM_LIGHTS_INDEX]      := ADR(DOWNSTAIRS_BEDROOM_LIGHTS_IN);
        LIGHTS_INPUTS[C_KITCHEN_LIGHTS_INDEX]              := ADR(KITCHEN_LIGHTS_IN);
        LIGHTS_INPUTS[C_DINING_ROOM_LIGHTS_INDEX]              := ADR(DINING_ROOM_LIGHTS_IN);
        LIGHTS_INPUTS[C_LIVING_ROOM_LIGHTS_INDEX]             := ADR(LIVING_ROOM_LIGHTS_IN);
        LIGHTS_INPUTS[C_TERRACE_LIGHTS_INDEX]              := ADR(TERRACE_LIGHTS_IN);
        LIGHTS_INPUTS[C_HALLWAY_LIGHTS_INDEX]             := ADR(HALLWAY_LIGHTS_COMBINED_IN);
        LIGHTS_INPUTS[C_BOILER_LIGHTS_INDEX]               := ADR(BOILER_LIGHTS_IN);
//        LIGHTS_INPUTS[C_STAIRS_LIGHTS_INDEX]              := ADR(STAIRS_LIGHTS_IN);

        LIGHTS_OUTPUTS[C_DOWNSTAIRS_BATH_MAJOR_LIGHTS_INDEX]     := ADR(DOWNSTAIRS_BATH_MAJOR_LIGHTS_OUT);
        LIGHTS_OUTPUTS[C_DOWNSTAIRS_BATH_SHOWER_LIGHTS_INDEX]   := ADR(DOWNSTAIRS_BATH_SHOWER_LIGHTS_OUT);
        LIGHTS_OUTPUTS[C_UPSTAIRS_BATH_MAJOR_LIGHTS_INDEX]    := ADR(UPSTAIRS_BATH_MAJOR_LIGHTS_OUT);
        LIGHTS_OUTPUTS[C_UPSTAIRS_WC_LIGHTS_INDEX]            := ADR(UPSTAIRS_WC_LIGHTS_OUT);
        LIGHTS_OUTPUTS[C_UPSTAIRS_BATH_SHOWER_LIGHTS_INDEX]  := ADR(UPSTAIRS_BATH_SHOWER_LIGHTS_OUT);
        LIGHTS_OUTPUTS[C_OUTDOOR_LIGHTS_INDEX]             := ADR(OUTDOOR_LIGHTS_OUT);
        LIGHTS_OUTPUTS[C_HALL_LIGHTS_INDEX]            := ADR(HALL_LIGHTS_OUT);
        LIGHTS_OUTPUTS[C_GARAGE_LIGHTS_INDEX]              := ADR(GARAGE_LIGHTS_OUT);
        LIGHTS_OUTPUTS[C_MAJOR_STORAGE_LIGHTS_INDEX]         := ADR(MAJOR_STORAGE_LIGHTS_OUT);
        LIGHTS_OUTPUTS[C_MINOR_STORAGE_LIGHTS_INDEX]          := ADR(MINOR_STORAGE_LIGHTS_OUT);
        LIGHTS_OUTPUTS[C_GARDEN_BALCONY_LIGHTS_INDEX]        := ADR(GARDEN_BALCONY_LIGHTS_OUT);
        LIGHTS_OUTPUTS[C_CHILDRENS_ROOM_2_LIGHTS_INDEX]       := ADR(CHILDRENS_ROOM_2_LIGHTS_OUT);
        LIGHTS_OUTPUTS[C_CHILDRENS_ROOM_1_OUTER_LIGHTS_INDEX] := ADR(CHILDRENS_ROOM_1_OUTER_LIGHTS_OUT);
        LIGHTS_OUTPUTS[C_CHILDRENS_ROOM_1_INNER_LIGHTS_INDEX] := ADR(CHILDRENS_ROOM_1_INNER_LIGHTS_OUT);
        LIGHTS_OUTPUTS[C_CHILDRENS_ROOM_3_LIGHTS_INDEX]       := ADR(CHILDRENS_ROOM_3_LIGHTS_OUT);
        LIGHTS_OUTPUTS[C_GATE_BALCONY_LIGHTS_INDEX]         := ADR(GATE_BALCONY_LIGHTS_OUT);
        LIGHTS_OUTPUTS[C_DOWNSTAIRS_BEDROOM_LIGHTS_INDEX]      := ADR(DOWNSTAIRS_BEDROOM_LIGHTS_OUT);
        LIGHTS_OUTPUTS[C_KITCHEN_LIGHTS_INDEX]              := ADR(KITCHEN_LIGHTS_OUT);
        LIGHTS_OUTPUTS[C_DINING_ROOM_LIGHTS_INDEX]              := ADR(DINING_ROOM_LIGHTS_OUT);
        LIGHTS_OUTPUTS[C_LIVING_ROOM_LIGHTS_INDEX]             := ADR(LIVING_ROOM_LIGHTS_OUT);
        LIGHTS_OUTPUTS[C_TERRACE_LIGHTS_INDEX]              := ADR(TERRACE_LIGHTS_OUT);
        LIGHTS_OUTPUTS[C_HALLWAY_LIGHTS_INDEX]             := ADR(HALLWAY_LIGHTS_OUT);
        LIGHTS_OUTPUTS[C_BOILER_LIGHTS_INDEX]               := ADR(BOILER_LIGHTS_OUT);
//        LIGHTS_OUTPUTS[C_STAIRS_LIGHTS_INDEX]              := ADR(HALLWAY_LIGHTS_OUT);

        LIGHTS_NAMES[C_DOWNSTAIRS_BATH_MAJOR_LIGHTS_INDEX]     := 'DOWNSTAIRS_BATH_MAJOR_LIGHTS';
        LIGHTS_NAMES[C_DOWNSTAIRS_BATH_SHOWER_LIGHTS_INDEX]   := 'DOWNSTAIRS_BATH_SHOWER_LIGHTS';
        LIGHTS_NAMES[C_UPSTAIRS_BATH_MAJOR_LIGHTS_INDEX]    := 'UPSTAIRS_BATH_MAJOR_LIGHTS';
        LIGHTS_NAMES[C_UPSTAIRS_WC_LIGHTS_INDEX]            := 'UPSTAIRS_WC_LIGHTS';
        LIGHTS_NAMES[C_UPSTAIRS_BATH_SHOWER_LIGHTS_INDEX]  := 'UPSTAIRS_BATH_SHOWER_LIGHTS';
        LIGHTS_NAMES[C_OUTDOOR_LIGHTS_INDEX]             := 'OUTDOOR_LIGHTS';
        LIGHTS_NAMES[C_HALL_LIGHTS_INDEX]            := 'HALL_LIGHTS';
        LIGHTS_NAMES[C_GARAGE_LIGHTS_INDEX]              := 'GARAGE_LIGHTS';
        LIGHTS_NAMES[C_MAJOR_STORAGE_LIGHTS_INDEX]         := 'MAJOR_STORAGE_LIGHTS';
        LIGHTS_NAMES[C_MINOR_STORAGE_LIGHTS_INDEX]          := 'MINOR_STORAGE_LIGHTS';
        LIGHTS_NAMES[C_GARDEN_BALCONY_LIGHTS_INDEX]        := 'GARDEN_BALCONY_LIGHTS';
        LIGHTS_NAMES[C_CHILDRENS_ROOM_2_LIGHTS_INDEX]       := 'CHILDRENS_ROOM_2_LIGHTS';
        LIGHTS_NAMES[C_CHILDRENS_ROOM_1_OUTER_LIGHTS_INDEX] := 'CHILDRENS_ROOM_1_OUTER_LIGHTS';
        LIGHTS_NAMES[C_CHILDRENS_ROOM_1_INNER_LIGHTS_INDEX] := 'CHILDRENS_ROOM_1_INNER_LIGHTS';
        LIGHTS_NAMES[C_CHILDRENS_ROOM_3_LIGHTS_INDEX]       := 'CHILDRENS_ROOM_3_LIGHTS';
        LIGHTS_NAMES[C_GATE_BALCONY_LIGHTS_INDEX]         := 'GATE_BALCONY_LIGHTS';
        LIGHTS_NAMES[C_DOWNSTAIRS_BEDROOM_LIGHTS_INDEX]      := 'DOWNSTAIRS_BEDROOM_LIGHTS';
        LIGHTS_NAMES[C_KITCHEN_LIGHTS_INDEX]              := 'KITCHEN_LIGHTS';
        LIGHTS_NAMES[C_DINING_ROOM_LIGHTS_INDEX]              := 'DINING_ROOM_LIGHTS';
        LIGHTS_NAMES[C_LIVING_ROOM_LIGHTS_INDEX]             := 'LIVING_ROOM_LIGHTS';
        LIGHTS_NAMES[C_TERRACE_LIGHTS_INDEX]              := 'TERRACE_LIGHTS';
        LIGHTS_NAMES[C_HALLWAY_LIGHTS_INDEX]             := 'HALLWAY_LIGHTS';
        LIGHTS_NAMES[C_BOILER_LIGHTS_INDEX]               := 'BOILER_LIGHTS';
//        LIGHTS_NAMES[C_STAIRS_LIGHTS_INDEX]              := 'STAIRS_LIGHTS_DOWNSTAIRS';

        VIRTUAL_LIGHTS_INPUTS[C_DOWNSTAIRS_BATH_MAJOR_LIGHTS_INDEX]     := ADR(VIRTUAL_DOWNSTAIRS_BATH_MAJOR_LIGHTS_IN);
        VIRTUAL_LIGHTS_INPUTS[C_DOWNSTAIRS_BATH_SHOWER_LIGHTS_INDEX]   := ADR(VIRTUAL_DOWNSTAIRS_BATH_SHOWER_LIGHTS_IN);
        VIRTUAL_LIGHTS_INPUTS[C_UPSTAIRS_BATH_MAJOR_LIGHTS_INDEX]    := ADR(VIRTUAL_UPSTAIRS_BATH_MAJOR_LIGHTS_IN);
        VIRTUAL_LIGHTS_INPUTS[C_UPSTAIRS_WC_LIGHTS_INDEX]            := ADR(VIRTUAL_UPSTAIRS_WC_LIGHTS_IN);
        VIRTUAL_LIGHTS_INPUTS[C_UPSTAIRS_BATH_SHOWER_LIGHTS_INDEX]  := ADR(VIRTUAL_UPSTAIRS_BATH_SHOWER_LIGHTS_IN);
        VIRTUAL_LIGHTS_INPUTS[C_OUTDOOR_LIGHTS_INDEX]             := ADR(VIRTUAL_OUTDOOR_LIGHTS_IN);
        VIRTUAL_LIGHTS_INPUTS[C_HALL_LIGHTS_INDEX]            := ADR(VIRTUAL_HALL_LIGHTS_IN);
        VIRTUAL_LIGHTS_INPUTS[C_GARAGE_LIGHTS_INDEX]              := ADR(VIRTUAL_GARAGE_LIGHTS_IN);
        VIRTUAL_LIGHTS_INPUTS[C_MAJOR_STORAGE_LIGHTS_INDEX]         := ADR(VIRTUAL_MAJOR_STORAGE_LIGHTS_IN);
        VIRTUAL_LIGHTS_INPUTS[C_MINOR_STORAGE_LIGHTS_INDEX]          := ADR(VIRTUAL_MINOR_STORAGE_LIGHTS_IN);
        VIRTUAL_LIGHTS_INPUTS[C_GARDEN_BALCONY_LIGHTS_INDEX]        := ADR(VIRTUAL_GARDEN_BALCONY_LIGHTS_IN);
        VIRTUAL_LIGHTS_INPUTS[C_CHILDRENS_ROOM_2_LIGHTS_INDEX]       := ADR(VIRTUAL_CHILDRENS_ROOM_2_LIGHTS_IN);
        VIRTUAL_LIGHTS_INPUTS[C_CHILDRENS_ROOM_1_OUTER_LIGHTS_INDEX] := ADR(VIRTUAL_CHILDRENS_ROOM_1_OUTER_LIGHTS_IN);
        VIRTUAL_LIGHTS_INPUTS[C_CHILDRENS_ROOM_1_INNER_LIGHTS_INDEX] := ADR(VIRTUAL_CHILDRENS_ROOM_1_INNER_LIGHTS_IN);
        VIRTUAL_LIGHTS_INPUTS[C_CHILDRENS_ROOM_3_LIGHTS_INDEX]       := ADR(VIRTUAL_CHILDRENS_ROOM_3_LIGHTS_IN);
        VIRTUAL_LIGHTS_INPUTS[C_GATE_BALCONY_LIGHTS_INDEX]         := ADR(VIRTUAL_GATE_BALCONY_LIGHTS_IN);
        VIRTUAL_LIGHTS_INPUTS[C_DOWNSTAIRS_BEDROOM_LIGHTS_INDEX]      := ADR(VIRTUAL_DOWNSTAIRS_BEDROOM_LIGHTS_IN);
        VIRTUAL_LIGHTS_INPUTS[C_KITCHEN_LIGHTS_INDEX]              := ADR(VIRTUAL_KITCHEN_LIGHTS_IN);
        VIRTUAL_LIGHTS_INPUTS[C_DINING_ROOM_LIGHTS_INDEX]              := ADR(VIRTUAL_DINING_ROOM_LIGHTS_IN);
        VIRTUAL_LIGHTS_INPUTS[C_LIVING_ROOM_LIGHTS_INDEX]             := ADR(VIRTUAL_LIVING_ROOM_LIGHTS_IN);
        VIRTUAL_LIGHTS_INPUTS[C_TERRACE_LIGHTS_INDEX]              := ADR(VIRTUAL_TERRACE_LIGHTS_IN);
        VIRTUAL_LIGHTS_INPUTS[C_HALLWAY_LIGHTS_INDEX]             := ADR(VIRTUAL_HALLWAY_LIGHTS_IN);
        VIRTUAL_LIGHTS_INPUTS[C_BOILER_LIGHTS_INDEX]               := ADR(VIRTUAL_BOILER_LIGHTS_IN);
//        VIRTUAL_LIGHTS_INPUTS[C_STAIRS_LIGHTS_INDEX]              := ADR(VIRTUAL_STAIRS_LIGHTS_IN);
    ELSE
        // No operation
    END_IF;

END_PROGRAM

(* ---- PersistData.ST ---- *)
PROGRAM PersistData
  VAR_INPUT
  END_VAR
  VAR_OUTPUT
  END_VAR
  VAR
    init : BOOL := FALSE;
    realPersistors : ARRAY [1 .. C_REALS_TO_PERSIST] OF PersistReal;
    boolPersistors : ARRAY [1 .. C_BOOLS_TO_PERSIST] OF PersistBool;

    i: INT := 0;
  END_VAR
  VAR_TEMP
  END_VAR

  FOR i := 1 to C_REALS_TO_PERSIST DO
    realPersistors[i](compilerBugPlaceholder := init,
      variableToPersist := REALS_TO_PERSIST[i]^,
      dirPath := REALS_TO_PERSIST_DIRS[i],
      fileName := REALS_TO_PERSIST_NAMES[i],
      toWrite := init);
  END_FOR;

  FOR i := 1 to C_BOOLS_TO_PERSIST DO
    boolPersistors[i](compilerBugPlaceholder := init,
      variableToPersist := BOOLS_TO_PERSIST[i]^,
      dirPath := BOOLS_TO_PERSIST_DIRS[i],
      fileName := BOOLS_TO_PERSIST_NAMES[i],
      toWrite := init);
  END_FOR;

  init := TRUE;

END_PROGRAM

(* ---- PersistInit.st ---- *)
PROGRAM PersistInit
  VAR_INPUT
  END_VAR
  VAR_OUTPUT
  END_VAR
  VAR
    init : BOOL := FALSE;
    i : INT := 0;
    ipidPath : STRING;
    heatingRootPath : STRING;
    roomTempPath : STRING;
    boilerControlPath : STRING;
  END_VAR
  VAR_TEMP
  END_VAR

  ipidPath := CONCAT(C_PERSIST_DIRECTORY_ROOT, C_PERSIST_HEATING_IPID_SUBDIR);
  heatingRootPath := CONCAT(C_PERSIST_DIRECTORY_ROOT, C_PERSIST_HEATING_SUBDIR);
  roomTempPath := CONCAT(heatingRootPath, C_PERSIST_ROOM_TEMPERATURE_SUBDIR);
  boilerControlPath := CONCAT(heatingRootPath, C_PERSIST_BOILER_CONTROL_SUBDIR);

  createDirectory(dirPath := C_PERSIST_DIRECTORY_ROOT);
    createDirectory(dirPath := ipidPath);
    createDirectory(dirPath := heatingRootPath);
        createDirectory(dirPath := roomTempPath);
        createDirectory(dirPath := boilerControlPath);

  IF NOT init THEN
    FOR i := 1 TO C_HEATING_ZONES DO
      REALS_TO_PERSIST[i] := DESIRED_TEMPERATURES[i-1];
      REALS_TO_PERSIST_NAMES[i] := INT_TO_STRING(i);
      REALS_TO_PERSIST_DIRS[i] := roomTempPath;
    END_FOR;

    REALS_TO_PERSIST[C_HEATING_ZONES + 1]        := ADR(IPID_K);
    REALS_TO_PERSIST_NAMES[C_HEATING_ZONES + 1]  := 'IPIDK';
    REALS_TO_PERSIST_DIRS[C_HEATING_ZONES + 1]   := boilerControlPath;
    REALS_TO_PERSIST[C_HEATING_ZONES + 2]        := ADR(IPID_TD);
    REALS_TO_PERSIST_NAMES[C_HEATING_ZONES + 2]  := 'IPIDTD';
    REALS_TO_PERSIST_DIRS[C_HEATING_ZONES + 2]   := boilerControlPath;
    REALS_TO_PERSIST[C_HEATING_ZONES + 3]        := ADR(IPID_TI);
    REALS_TO_PERSIST_NAMES[C_HEATING_ZONES + 3]  := 'IPIDTI';
    REALS_TO_PERSIST_DIRS[C_HEATING_ZONES + 3]   := boilerControlPath;
    REALS_TO_PERSIST[C_HEATING_ZONES + 4]        := ADR(OVERSHOOT_HISTERESIS);
    REALS_TO_PERSIST_NAMES[C_HEATING_ZONES + 4]  := 'OVHISTER';
    REALS_TO_PERSIST_DIRS[C_HEATING_ZONES + 4]   := boilerControlPath;

    BOOLS_TO_PERSIST[1]       := ADR(HEATING_ENABLE);
    BOOLS_TO_PERSIST_NAMES[1] := 'BOILER';
    BOOLS_TO_PERSIST_DIRS[1]  := boilerControlPath;
    BOOLS_TO_PERSIST[2]       := ADR(HOT_WATER_ENABLE);
    BOOLS_TO_PERSIST_DIRS[2]  := boilerControlPath;
    BOOLS_TO_PERSIST_NAMES[2] := 'HOTWATER';
    BOOLS_TO_PERSIST[3]       := ADR(PRESENCE_BASED_HEATING_CONTROL);
    BOOLS_TO_PERSIST_NAMES[3] := 'PRESENCE_BOILER_CONTROL';
    BOOLS_TO_PERSIST_DIRS[3]  := boilerControlPath;
    BOOLS_TO_PERSIST[4]       := ADR(PRESENCE_BASED_HOT_WATER_ENABLE);
    BOOLS_TO_PERSIST_DIRS[4]  := boilerControlPath;
    BOOLS_TO_PERSIST_NAMES[4] := 'PRESENCE_HOTWATER_CONTROL';
    init := TRUE;

  ELSE
    // No operation
  END_IF;

END_PROGRAM

(* ---- WateringInit.ST ---- *)
PROGRAM WateringInit
  VAR_INPUT
  END_VAR
  VAR_OUTPUT
  END_VAR
  VAR
  END_VAR
  VAR_TEMP
  END_VAR

END_PROGRAM
